(* ---------------------- Debug-Message ----------------------------*)
(*IF  _debug_enable THEN
	IF state <> state_last THEN
		LOG_CL.NEW_MSG := 'IP_STEP ~1 -IP_ID ~6';
		LOG_CL.PRINTF[1] := BYTE_TO_STRING(state);
		LOG_CL.PRINTF[6] := INT_TO_STRING(debug_ID);
		LOG_MSG();
		state_last := state;
	END_IF;
END_IF;*)
(* -----------------------------------------------------------------------------*)

IF IP_C.TIME_RESET THEN (* Alle Timer ruecksetzen *)
	IP_C.TIME_RESET := FALSE; (* Reset rücksetzen *)
	c_time := tx; (* Connect Timer ruecksetzen *)
	s_time := tx; (* Send Timer ruecksetzen *)
	r_time := tx; (* Receive Timer ruecksetzen *)

	c_status := BYTE#0; (* letzten Connect Fehler rücksetzen *)
	s_status := BYTE#0; (* letzten Send Fehler rücksetzen *)
	r_status := BYTE#0; (* letzten Receive Fehler rücksetzen *)
END_IF;

(* ---------------------------------------------- *)

CASE state OF

UDP_INIT: (* UDP_CLIENT + SERVER *)
	socket := SysSockCreate(SOCKET_AF_INET, SOCKET_DGRAM, SOCKET_IPPROTO_IP, ADR(pResult));
	IF socket < 0 THEN
		c_status := 1; (* SysSockCreate failed *)
		state := C_CLOSE;
	ELSE
		FunctionResult :=SysSockSetOption(socket, SOCKET_SOL, SOCKET_SO_BROADCAST, ADR(dint_true), SIZEOF(dint_true)); (* allow broadcast *)
		FunctionResult :=SysSockIoctl(socket, SOCKET_FIONBIO, ADR(dint_true)); (* put socket in non-blocking mode *)
		sockaddr.sin_family := SOCKET_AF_INET;
		sockaddr.sin_port := SysSockHtons(c_port);
		sockaddr.sin_addr.ulAddr := SEL(c_mode = 1, SOCKET_INADDR_ANY, SysSockNtohl(c_ip));

		IF c_mode >= 2 THEN (* SERVER Mode *)
			FunctionResult := SysSockBind(socket, ADR(sockaddr), SIZEOF(sockaddr));
			IF FunctionResult=0 THEN
				c_ready := TRUE; (* Connected *)
				state:= C_WAIT;
			ELSE
				c_status := 2; (* SysSockBind failed *)
				state := C_CLOSE;
			END_IF;
		ELSE
			c_ready := TRUE; (* Connected *)
			state:= C_WAIT;
		END_IF;
	END_IF;

(* ---------------------------------------------- *)

TC_INIT: (* TCP-CLIENT (AKTIV) *)
	// Create handle to ethernet socket to send messages
	socket        := SysSockCreate(SOCKET_AF_INET, SOCKET_STREAM, SOCKET_IPPROTO_TCP, ADR(pResult)); 	
	IF socket < 0 THEN
		c_status := 1;  (* SysSockCreate failed *)
		state := C_CLOSE;
	ELSE
		IF plc_841 OR plc_881 THEN
			FunctionResult :=SysSockSetOption(socket,6,SOCKET_TCP_NODELAY, ADR(dint_true), SIZEOF(dint_true)); (* Set Push-Bit *)
		END_IF;
		// Set option for local address reuse
		FunctionResult :=SysSockSetOption(socket, SOCKET_SOL, SOCKET_SO_REUSEADDR, ADR(dint_true), SIZEOF(dint_true));
		// Set option for keepalive
		//FunctionResult := SysSockSetOption(socket, SOCKET_SOL, SOCKET_SO_KEEPALIVE, ADR(dint_true), SIZEOF(dint_true));
		
        FunctionResult :=SysSockIoctl(socket, SOCKET_FIONBIO, ADR(dint_true)); (* NonBlocking mode *)
		
		sockaddr.sin_family := SOCKET_AF_INET;
		sockaddr.sin_port := SysSockNtohs(c_port);
		sockaddr.sin_addr.ulAddr  := SysSockNtohl(c_ip);
		c_select := FALSE;
		state := TC_CONNECT;
	END_IF;

(* ---------------------------------------------- *)

TC_CONNECT:
	IF NOT c_enable OR c_status = 255 THEN (* keine freigabe oder connect timeout *)
			state:= C_CLOSE;
	ELSE
		IF c_select = FALSE THEN
			FunctionResult:=SysSockConnect(socket,ADR(sockaddr),SIZEOF(sockaddr));
			IF FunctionResult=0 THEN
				c_ready := TRUE; (* Connected *)
				state:= C_WAIT;
			ELSE
				(* Connect durchgeführt, aber noch nicht verbunden, dann optional mit select-abfrage weitermachen *)
				c_select := SYSLIBSOCKETS_OPTION.0; (* Bit 0 = TCP-Client - use SysSockselect *)
			END_IF;
		ELSE
			c_Timeout.tv_sec := 0;
			c_Timeout.tv_usec := 0;
			c_fdWrite.fd_count := 1;
			c_fdWrite.fd_array[0] := socket;
			IF SysSockSelect(SOCKET_FD_SETSIZE,0,ADR(c_fdWrite),0, ADR(c_Timeout), ADR(pResult)) > 0 THEN
				c_ready := TRUE; (* Connected *)
				state:= C_WAIT;
			END_IF;
		END_IF;
	END_IF;

(* ---------------------------------------------- *)

TS_INIT: (* TCP-SERVER (PASSIV) *)
	server_socket := SysSockCreate(SOCKET_AF_INET, SOCKET_STREAM, SOCKET_IPPROTO_IP, ADR(pResult)); (* Create Socket *)
	IF server_socket = RTS_INVALID_HANDLE THEN
		c_status := 1; (* SysSockCreate failed *)
		state:= C_CLOSE;
	ELSE (* Address bindings *)
		SysSockSetOption( server_socket, SOCKET_SOL, SOCKET_SO_REUSEADDR, ADR(dint_true), SIZEOF(dint_true) );
		sockaddr.sin_family:= SOCKET_AF_INET;
		sockaddr.sin_port := SysSockHtons(c_port);
		sockaddr.sin_addr.ulAddr  := SOCKET_INADDR_ANY;
		IF NOT SysSockBind(server_socket, ADR(sockaddr), SIZEOF(sockaddr)) = 0 THEN
			c_status := 2; (* SysSockBind failed *)
			state := C_CLOSE;
		ELSIF NOT SysSockListen(server_socket, 1) = 0 THEN (* erzeugt Warteschlange für eine Verbindung *)
			c_status := 3; (* SysSockListen failed *)
			state:= C_CLOSE;
		ELSE
			SysSockIoctl(server_socket, SOCKET_FIONBIO, ADR(dint_true)); (* NonBlocking mode *)
			state:= TS_OPEN;
		END_IF;
	END_IF;

(* ---------------------------------------------- *)

TS_OPEN: (* Waiting for incomming connection *)
	sockaddr_size := SIZEOF(sockaddr);
	socket := SysSockAccept(server_socket, ADR(sockaddr), ADR(sockaddr_size), ADR(pResult));

	IF socket <> RTS_INVALID_HANDLE THEN (* neuer Verbindungswunsch vorhanden *)
		IF c_mode = BYTE#2 AND sockaddr.sin_addr.ulAddr <> SysSockNtohl(c_ip) THEN (* Mode 2 = TCP + PASSIVE + PORT + IP  auf richtige Partner-IP prüfen *)
			state:= C_CLOSE;
		ELSE
			IF plc_841 OR plc_881 THEN
				SysSockSetOption(socket, 6, SOCKET_TCP_NODELAY, ADR(dint_true), SIZEOF(dint_true)); (* Set Push-Bit *)
			END_IF;
			SysSockIoctl(socket, SOCKET_FIONBIO, ADR(dint_true)); (* NonBlocking mode *)
			c_ready := TRUE; (* Connected *)
			state := C_WAIT;
		END_IF;
	ELSIF NOT c_enable THEN (* keine freigabe mehr ? *)
			state:= C_CLOSE;
	END_IF;

(* ---------------------------------------------- *)

C_WAIT: (* Warten auf Anforderung für Beenden *)
	IF NOT c_enable OR NOT c_ready THEN
		state:= C_CLOSE;
	END_IF

(* ---------------------------------------------- *)

C_CLOSE: (* Close the Sockets *)
	c_ready := FALSE;
	IF socket >= 0 THEN
		IF (NOT plc_841) AND (NOT plc_881) THEN
			SysSockShutdown(socket, 0); (* 870 *)
		END_IF;
		SysSockClose(socket);
		socket := RTS_INVALID_HANDLE;
	END_IF
	IF server_socket >= 0 THEN
		IF (NOT plc_841) AND (NOT plc_881) THEN
			SysSockShutdown(server_socket, 0); (* 870 *)
		END_IF;
		SysSockClose(server_socket);
		server_socket := RTS_INVALID_HANDLE;
	END_IF
	state:= STOP;
END_CASE;

(* ---------------------------------------------- *)

IF c_ready THEN
	IF NOT c_ready_old THEN (* Verbindung aufgebaut - positive Flanke erkannt *)
		IP_C.C_STATE := 254;
		IP_C.TIME_RESET := TRUE; (* Alle Timer ruecksetzen *)
		(* ---------------------- Debug-Message ----------------------------*)
		(*IF _debug_enable THEN
			LOG_CL.NEW_MSG := 'IP_CON: CONNECTED -IP_ID ~6';
			LOG_CL.PRINTF[6] := INT_TO_STRING(debug_ID);
			LOG_MSG();
		END_IF;*)
		(* -----------------------------------------------------------------------------*)
	ELSE
		IP_C.C_STATE := 255; (* Verbindung ist aufgebaut *)
	END_IF;
ELSE
	IF c_ready_old THEN (* Verbindung abgebaut - negative Flanke erkannt *)
		IP_C.C_STATE := 1;
		IP_C.MAILBOX[1] := 0; (* Receive Info rücksetzen *)
		IP_C.MAILBOX[2] := 0; (* Send-Pause rücksetzen *)
		IP_C.MAILBOX[3] := 0; (* Receive-Pause rücksetzen *)
		IF NOT new_connection THEN
			s_active := FALSE; (* Sendeaktivitäten stoppen *)
			s_req := FALSE; (* Sendefreigabe rücksetzen *)
			S_BUF.SIZE := 0; (* Sendelänge löschen *)
			(*IP_C.TIME_RESET := TRUE;*) (* Alle Timer ruecksetzen *)
		END_IF;
		(* ---------------------- Debug-Message ----------------------------*)
		(*IF _debug_enable THEN
			LOG_CL.NEW_MSG := 'IP_CON: DISCONNECTED';
			LOG_MSG();
		END_IF;*)
		(* -----------------------------------------------------------------------------*)
	ELSE
		IP_C.C_STATE := 0; (* Verbindung ist abgebaut *)
	END_IF;
END_IF;

c_ready_old := c_ready;

(* Der Datenempfang wird angehalten solange ein Sendevorgang läuft *)
(* sonst kann es vorkommen das die Antwort-daten schon empfangen werden, *)
(* bevor der Sendevorgang vom programm abgeschlossen wurde *)

IF c_ready AND NOT s_active AND IP_C.MAILBOX[3] = 0 THEN
	IF R_BUF.SIZE >= INT_TO_UINT(r_max_size) THEN
		R_BUF.SIZE := UINT#0;
		r_status := 254; (* Empfangsbuffer wegen Überlauf rückgesetzt *)
	END_IF;

	r_offset := SEL(udp_mode,UINT_TO_INT(R_BUF.SIZE),0);
	r_count := r_max_size - r_offset;

	IF udp_mode THEN
		bytes_received := SysSockRecvFrom(socket, ADR(R_BUF.BUFFER), r_count, 0, ADR(sockaddr), SIZEOF(sockaddr), ADR(pResult));

		IF c_mode = BYTE#3 AND sockaddr.sin_addr.ulAddr <> SysSockNtohl(c_ip) THEN (* Mode 3 = UDP + PASSIVE + PORT + IP  auf richtige Partner-IP prüfen *)
			bytes_received := 0;
			R_BUF.SIZE := UINT#0;
			sockaddr.sin_port := SysSockNtohs(c_port);
			sockaddr.sin_addr.ulAddr  := SysSockNtohl(c_ip);
		END_IF;

	ELSE
		bytes_received := SysSockRecv(socket, ADR(R_BUF.BUFFER[r_offset]), r_count, 0, ADR(pResult));
	END_IF;

	CASE pResult OF
		518:  bytes_received:=-1; //Connection OKAY just no data and do not want to BIND
		521:  bytes_received:=0; //Connection has been refused by the remote host 
		523:  bytes_received:=0; //The host has not been found  
		524:  bytes_received:=0; //Host is unreachable  
		526:  bytes_received:=0; //The socket is not connected  
		527:  bytes_received:=0; //Shutdown has been called on the socket  
		529:  bytes_received:=0; //Socket has been gracefully closed. No more send/receives allowed	 
	END_CASE

	
	(*UDP: IPC returns -1 if no data available or error occured,841 returns -1 if error occured and 0 if no data available*)
	CASE bytes_received OF
	-2147483648..-1: ; (* No data available or error occured *)
	 0: IF NOT udp_mode OR pResult<>518 THEN (* TCP-Mode: socket wurde von remote geschlossen *)
			c_status := 253;
			c_ready := FALSE;
		END_IF;
	ELSE (* daten wurden empfangen *)
  		r_time := tx; (* Receive Timer ruecksetzen *)
		R_BUF.SIZE := INT_TO_UINT(r_offset) + DINT_TO_UINT(bytes_received); (* aktuelle buffersize eintragen *)
		IP_C.MAILBOX[1] := IP_C.MAILBOX[1] + 1; (* Receive Info *)
		IF IP_C.MAILBOX[1] = 0 THEN IP_C.MAILBOX[1] := 1; END_IF;

		(* ---------------------- Debug-Message ----------------------------*)
		(*IF _debug_enable THEN
			LOG_CL.NEW_MSG := 'IP_REC DATA: POS: ~1 : SIZE: ~2 TOTAL ~3 -IP_ID ~6';
			LOG_CL.PRINTF[1] := INT_TO_STRING(r_offset);
			LOG_CL.PRINTF[2] := INT_TO_STRING(r_count);
			LOG_CL.PRINTF[3] := UINT_TO_STRING(R_BUF.SIZE);
			LOG_CL.PRINTF[6] := INT_TO_STRING(debug_ID);
			LOG_MSG();
		END_IF;*)
		(* -----------------------------------------------------------------------------*)

	END_CASE
END_IF;

(* ---------------------------------------------- *)

IF S_BUF.SIZE > 0 THEN
	IF c_ready AND c_enable THEN
		IF NOT s_active AND IP_C.MAILBOX[2] = 0 THEN
			(* Gesamtanzahl an Bytes limitieren und uebergeben *)
			s_total := LIMIT(0,UINT_TO_INT(S_BUF.SIZE),r_max_size);
			s_cur_pos  := 0;
			s_cur_size := 0;
			s_start := TRUE; (* Daten kopieren und senden anstossen *)
			s_active := TRUE; (* Sende-Betrieb aktivieren *)
			(* ---------------------- Debug-Message ----------------------------*)
			(*IF _debug_enable THEN
				LOG_CL.NEW_MSG := 'IP_SEN INIT: TOTAL: ~1 -IP_ID ~6';
				LOG_CL.PRINTF[1] := INT_TO_STRING(S_TOTAL);
				LOG_CL.PRINTF[6] := INT_TO_STRING(debug_ID);
				LOG_MSG();
			END_IF;*)
			(* -----------------------------------------------------------------------------*)
		END_IF;

		IF s_done OR s_start THEN (* Daten senden aktiv *)

			s_start := FALSE;
			s_cur_pos := s_cur_pos + s_cur_size; (* neue Sende-Datenposition bestimmen *)
			IF s_total > s_cur_pos THEN (* weitere Daten zum senden vorhanden ? *)
				s_cur_size := s_total - s_cur_pos;
				s_cur_size := LIMIT(0, s_cur_size, s_max_size); (* Telegrammlänge begrenzen *)
				(* ---------------------- Debug-Message ----------------------------*)
				(*IF _debug_enable THEN
					LOG_CL.NEW_MSG := 'IP_SEN DATA: POS: ~1 : SIZE: ~2 TOTAL ~3 -IP_ID ~6';
					LOG_CL.PRINTF[1] := INT_TO_STRING(S_CUR_POS);
					LOG_CL.PRINTF[2] := INT_TO_STRING(S_CUR_SIZE);
					LOG_CL.PRINTF[3] := INT_TO_STRING(S_TOTAL);
					LOG_CL.PRINTF[6] := INT_TO_STRING(debug_ID);
					LOG_MSG();
				END_IF;*)
				(* -----------------------------------------------------------------------------*)
				s_time := tx; (* Send Timer ruecksetzen *)
				r_time := tx; (* Receive Timer ruecksetzen *)
				s_req := TRUE;

			ELSE
				(* keine weitere Sendedaten vorhanden -> Senden beenden *)
				s_req := FALSE;
				s_active := FALSE;
				S_BUF.SIZE := 0;
				(* ---------------------- Debug-Message ----------------------------*)
				(*IF _debug_enable THEN
					LOG_CL.NEW_MSG := 'IP_SEN FINISH -IP_ID ~6';
					LOG_CL.PRINTF[6] := INT_TO_STRING(debug_ID);
					LOG_MSG();
				END_IF;*)
				(* -----------------------------------------------------------------------------*)
			END_IF;
		END_IF;
	END_IF;
END_IF;

IF s_req THEN
	s_done := FALSE;
	IF udp_mode THEN
		bytes_sent := SysSockSendTo(socket, ADR(S_BUF.BUFFER[s_cur_pos]), s_cur_size, 0, ADR(sockaddr), SIZEOF(sockaddr), ADR(pResult));
	ELSE
		bytes_sent := SysSockSend(socket, ADR(S_BUF.BUFFER[s_cur_pos]), s_cur_size, 0, ADR(pResult));
	END_IF;

	CASE bytes_sent OF
	-2147483648..-1:	; (* ERROR: Noch nicht bereit um Daten aufzunehmen -> nächsten Zyklus wieder probieren *)
	 0: IF NOT udp_mode THEN (* TCP-Mode: socket wurde von remote geschlossen *)
			c_status := 253;
			c_ready := FALSE;
		END_IF;
	ELSE
		s_done := TRUE;
		s_cur_size := DINT_TO_INT(bytes_sent); (* Anzahl der wirklich versendeten Bytes übernehmen *)
		(* ---------------------- Debug-Message ----------------------------*)
		(*IF _debug_enable THEN
			LOG_CL.NEW_MSG := 'IP_SEN SEND_COUNT ~1 -IP_ID ~6';
			LOG_CL.PRINTF[1] := DINT_TO_STRING(s_cur_size);
			LOG_CL.PRINTF[6] := INT_TO_STRING(debug_ID);
			LOG_MSG();
		END_IF;*)
		(* -----------------------------------------------------------------------------*)
	END_CASE
END_IF;

(* ---------------------------------------------- *)

IF IP_C.R_OBSERVE = FALSE OR s_active THEN
    r_time := tx;
END_IF;

IF c_status = 0 AND tx - c_time > error_time AND c_enable AND NOT c_ready AND c_mode < 2 THEN (* Connect Timeout *)
	c_status := 255; (* Timeout-Fehler ausgeben *)
END_IF;
IF s_status = 0 AND tx - s_time > error_time AND s_active THEN (* Send Timeout *)
	s_status := 255; (* Timeout-Fehler ausgeben *)
END_IF;
IF r_status = 0 AND tx - r_time > error_time AND c_ready AND IP_C.R_OBSERVE THEN (* Receive Timeout *)
	r_status := 255; (* Timeout-Fehler ausgeben *)
END_IF;

IP_C.ERROR := OSCAT_BASIC.DWORD_OF_BYTE(c_status,s_status,r_status,0);

(* ---------------------- Debug-Message ----------------------------*)
(*IF  _debug_enable THEN
	IF (IP_C.ERROR <> debug_lasterror) THEN
		LOG_CL.NEW_MSG := 'IP_ERROR ~1 -IP_ID ~6';
		LOG_CL.PRINTF[1] := DWORD_TO_STRING(IP_C.ERROR);
		LOG_CL.PRINTF[6] := INT_TO_STRING(debug_ID);
		LOG_MSG();

		debug_lasterror := IP_C.ERROR;
		debug_last_id := debug_ID;
	END_IF;
END_IF;*)
(* -----------------------------------------------------------------------------*)

(* revision history
ks	18. oct. 2008	rev 1.0
	original version
ks	05. jan. 2009	rev 1.1
	zusätzlichen Parameter "Port" hinzugefügt, und Code bei Verbindungsaufbau angepasst
ks	28. feb. 2009	rev 1.2
	connect code angepasst und verkürzung der zyklen bei Send
ks	20. oct. 2009	rev 1.3
	network_buffer basis 0
ks	06. dec. 2009	rev 1.4
	receive_count MAILBOX[1]
ks	10. nov. 2010	rev 1.5
	send_pause MAILBOX[2] and receive_pause MAILBOX[3] 
ks	07. feb. 2011	rev 1.6
	Fehlercode 253 bei Remote-Verbindungsabbruch
ks	30. may. 2011	rev 1.7
	Fehler bei Empfangsüberwachung
ks	26. july. 2011	rev 1.8
	Error-Reset, diverse optimierungen 
ks	26. feb. 2012	rev 1.9
	Code-Optimierung für höhere kompatibilität

*)

END_FUNCTION_BLOCK

// Common/Function Blocks/TIME_DATE_IMPULS
FUNCTION_BLOCK TIME_DATE_IMPULS
VAR_IN_OUT
	TDI_Data:TIME_DATE_IMPULS_DATA;
END_VAR
VAR_INPUT
END_VAR

VAR
	RT_SYS:RTCLK.GetDateAndTime;
	RT:OSCAT_BASIC.RTC_2;
	DT_OLD:DT;
	GET_TIME: BOOL := TRUE;
	TIME_READED: BOOL;
	TIMEZONE:RTCLK.PERIODE;
	ReReadTime: BOOL;
	ReReadErrorTime:TON;
	ReReadTimeCycle:TON;
	DayChangeEdge:R_TRIG;
END_VAR

RT_SYS(xExecute := GET_TIME);
IF RT_SYS.xDone THEN
	GET_TIME := FALSE;
	IF	RT_SYS.dtDateAndTime < DT#1980-01-01-00:00:00 THEN
		//Keine Valide Uhr auf Raspi!
		ReReadTime := TRUE;
		TDI_Data.TIME_IO := FALSE;
	ELSE
		TIME_READED := TRUE;
		TIMEZONE := RT_SYS.eTimezone;
		ReReadTime := FALSE;
		TDI_Data.TIME_IO := TRUE;
	END_IF
END_IF
//Zykliches neulsesen der Uhrzeit
ReReadTimeCycle(in := (TDI_Data.TIME_IO AND NOT GET_TIME), PT:= T#30M);
IF ReReadTimeCycle.Q THEN
	GET_TIME := TRUE;//try again to read Time	
END_IF


//Neulesezeit nach Error bearbeiten:
ReReadErrorTime(in:=ReReadTime, pt:=T#1S);
IF ReReadErrorTime.Q THEN
	ReReadTime := FALSE;
	GET_TIME := TRUE;//try again to read Time
END_IF
//Realtime Clock bearbeiten // Setzten
RT(set := TIME_READED, SDT := RT_SYS.dtDateAndTime, OFS := 60, DEN:=TRUE,);
TIME_READED := FALSE;
//Date and time from oscat fb
TDI_Data.SYSTEM_TIME:=RT._LDT;
//check for second impuls
IF DT_OLD <> TDI_Data.SYSTEM_TIME THEN
	DT_OLD := TDI_Data.SYSTEM_TIME;
	TDI_Data.imp := TRUE;
ELSE
	TDI_Data.imp := FALSE;
END_IF
//make Time for OSCAT functions
TDI_Data.TD_TIME := OSCAT_BASIC.DT_TO_SDT(DTI:= TDI_Data.SYSTEM_TIME);
TDI_Data.UDT := RT.UDT;

DayChangeEdge(CLK:=TO_TOD(TDI_DATA.SYSTEM_TIME)= TOD#00:00:00);
TDI_DATA.DAY_CHANGE := DayChangeEdge.Q;

END_FUNCTION_BLOCK

// Common/Functions/GET_DNS_IP
FUNCTION GET_DNS_IP : STRING(16)
VAR_INPUT
END_VAR
VAR
	Result:RTS_IEC_RESULT;
	DNS_STRING:STRING(1000);
	findRet:DINT;
	i:INT;
	j:INT;
	k:INT;
	start:INT;
	stop:INT;
	//id of operating system
	OsId:UDINT;
END_VAR
VAR CONSTANT
	GET_DNS_COMMAND_LINUX:STRING:='cat /etc/resolv.conf ';//|grep -i nameserver|head -n1|cut -d $' $' -f2';
	GET_DNS_COMMAND_WINDOWS:STRING:='powershell Get-DnsClientServerAddress';//|grep -i nameserver|head -n1|cut -d $' $' -f2';
	NAMESERVER_LINUX:STRING:='nameserver';
	
END_VAR

(*
for linux

change 
sudo nano /etc/CODESYSControl.cfg
or from runtime version 4.5.11.20
sudo nano /etc/CODESYSControl_User.cfg 
[SysProcess]
Command.0=shutdown

to 

[SysProcess]
Command.0=shutdown
Command.1=cat

for windows, needs powershell

"C:\ProgramData\CODESYS\CODESYSControlWinV3\???\CODESYSControl.cfg"
[SysProcess]
BasePriority=Realtime
Command=AllowAll

*)

//cat /etc/resolv.conf |grep -i nameserver|head -n1|cut -d ' ' -f2
//get content

SysTargetGetOperatingSystemId(pudiOperatingSystemId:= ADR(OsId));


GET_DNS_IP := 'ERROR';

IF OsId = OperatingSystemID.SYSTARGET_OS_LINUX THEN

	SysProcess.SysProcessExecuteCommand2(pszCommand:=GET_DNS_COMMAND_LINUX,pszStdOut:= DNS_STRING,udiStdOutLen:=SIZEOF(DNS_STRING),pResult:=ADR(Result));
	IF Result = CmpErrors.Errors.ERR_NO_ACCESS_RIGHTS THEN
		GET_DNS_IP := 'NOACCESSRIGHTS';
		RETURN;
	END_IF
	//TODO check if command is enabled 
	i:= Standard.FIND(STR1:=DNS_STRING, STR2:=NAMESERVER_LINUX);
	IF i < 0 THEN RETURN; END_IF
	j := OSCAT_BASIC.FIND_CTRL(str:= DNS_STRING, pos:= i);
	IF j <= 0 THEN RETURN; END_IF
	
	GET_DNS_IP := Standard.MID(STR:= DNS_STRING, LEN:= j - i - Standard.LEN(STR:=NAMESERVER_LINUX) - 1, POS:= i + Standard.LEN(NAMESERVER_LINUX) + 1);
	
END_IF

IF OsId = OperatingSystemID.SYSTARGET_OS_WINDOWS THEN
{info 'TODO: hind that this is blocking!'}
SysProcess.SysProcessExecuteCommand2(pszCommand:=GET_DNS_COMMAND_WINDOWS,pszStdOut:= DNS_STRING,udiStdOutLen:=SIZEOF(DNS_STRING),pResult:=ADR(Result));
	IF Result = CmpErrors.Errors.ERR_NO_ACCESS_RIGHTS THEN
		GET_DNS_IP := 'NOACCESSRIGHTS';
		RETURN;
	END_IF
	//TODO check if command is enabled 
	findRet:= find(STR1:=ADR(DNS_STRING), STR2:=ADR('IPv4'));
	IF findRet < 0 THEN RETURN; END_IF
	i := DINT_TO_INT(findRet);
	//now search '{'
	FOR j := 0 TO 40 DO//max 40 chars space
		IF DNS_STRING[i + j] = GetChar('{') THEN
			start := i + j + 1;
		END_IF
 		IF DNS_STRING[i + j] = GetChar('}') THEN
			stop := i + j - 1;
			EXIT;
		END_IF
	END_FOR
	//now copy data, string functions usless --> more than 255 chars...
	
	j := 0;
	FOR i := start TO stop DO
		GET_DNS_IP[j] := DNS_STRING[i];
		j := j + 1;
	END_FOR
	GET_DNS_IP[j] := 0;//termination
	
	//j := OSCAT_BASIC.FIND_CTRL(str:= DNS_STRING, pos:= i);
//	IF j <= 0 THEN RETURN; END_IF
	
	//GET_DNS_IP := Standard.MID(STR:= DNS_STRING, LEN:= j - i - Standard.LEN(STR:=NAMESERVER_LINUX) - 1, POS:= i + Standard.LEN(NAMESERVER_LINUX) + 1);
	

END_IF

END_FUNCTION

// Common/Functions/find
//searchs str2 in str1
FUNCTION find : DINT
VAR_INPUT
	str1:POINTER TO STRING;
	str2:POINTER TO STRING;
END_VAR
VAR
	
	n:UINT;	
	pt:POINTER TO BYTE;
	
	j: UINT;
END_VAR

find := -1;//first we din't find anything....
n := len(str := str2);


pt := str1;

WHILE pt^ <> 0 DO
	IF SysMemCmp(pBuffer1:= pt, pBuffer2:= str2, udiCount:= n) = 0 THEN
		
		find := j;
		RETURN;
	
	END_IF
	j := j + 1;
	pt := pt + SIZEOF(BYTE);
	
END_WHILE

END_FUNCTION

// Common/Functions/len
FUNCTION len : UINT
VAR_INPUT
	str:POINTER TO STRING;
END_VAR
VAR
	k:uINT;
	pt:POINTER TO BYTE;
END_VAR

pt := str;
WHILE pt[k] <>  0 DO
	k := k + 1;
END_WHILE
len := k;

END_FUNCTION

// Common/Functions/GetChar
FUNCTION GetChar : byte
VAR_INPUT
	in:STRING(1);
END_VAR

GetChar := in[0];

END_FUNCTION

// Common/Functions/concat
FUNCTION concat : pointer to string
VAR_INPUT
	s1:POINTER TO STRING;
	s2:POINTER TO STRING;
END_VAR
VAR
	p1:POINTER TO BYTE;
	len1:UINT;
	
	ui:UINT;
END_VAR

p1 := ADR(s1^[len(s1)]);
len1 := len(s2);
SysMemMove(pDest:= p1, pSrc:= s2, udiCount:= len1 + 1);//+ 1 for add 0 to string end

concat := s1;

END_FUNCTION

// Common/Function Blocks/TestString
FUNCTION_BLOCK TestString 
VAR_INPUT
END_VAR
VAR
	s10:STRING:='1111111111';
	s102:STRING:='2222222222';
	sp:STRING(64000);
	ps1:POINTER TO STRING;
	lens:UINT;
END_VAR

lens := len(ADR(s10)); //needs to be 10!
sp:='';
concat(s1:= ADR(sp), s2:= ADR(s10));
ps1 := ADR(sp);
lens := len(ADR(sp)); //needs to be 10!

concat(s1:= ADR(sp), s2:= ADR(s102));

lens := len(ADR(sp)); //needs to be 20!

concat(s1:= ADR(sp), s2:= ADR(s10));

lens := len(ADR(sp)); //needs to be 30!

concat(s1:= ADR(sp), s2:= ADR(s102));

lens := len(ADR(sp)); //needs to be 40!

concat(s1:= ADR(sp), s2:= ADR(s10));

lens := len(ADR(sp)); //needs to be 50!

concat(s1:= ADR(sp), s2:= ADR(sp));

lens := len(ADR(sp)); //needs to be 100!

concat(s1:= ADR(sp), s2:= ADR(sp));

lens := len(ADR(sp)); //needs to be 200!

concat(s1:= ADR(sp), s2:= ADR(sp));

lens := len(ADR(sp)); //needs to be 400!

concat(s1:= ADR(sp), s2:= ADR(sp));

lens := len(ADR(sp)); //needs to be 800!

concat(s1:= ADR(sp), s2:= ADR(sp));

lens := len(ADR(sp)); //needs to be 1600!

concat(s1:= ADR(sp), s2:= ADR(sp));

lens := len(ADR(sp)); //needs to be 3200!

concat(s1:= ADR(sp), s2:= ADR(sp));

lens := len(ADR(sp)); //needs to be 6400!

END_FUNCTION_BLOCK

// Common/Function Blocks/IP_CONTROL_TLS
FUNCTION_BLOCK IP_CONTROL_TLS EXTENDS IP_CONTROL
VAR_INPUT
	TLS_CONFIG_IN:POINTER TO TLS_CONFIG := 0;(*info about tls stuff*)
	useTls: BOOL;

END_VAR
VAR_OUTPUT
END_VAR
VAR
	
END_VAR


TLS:= useTls;
IF TLS THEN
	TLS_CONFIG := TLS_CONFIG_IN;
END_IF
SUPER^(IP_C := IP_C, R_BUF:= R_BUF, S_BUF:= S_BUF);

END_FUNCTION_BLOCK

// Common/Functions/ResolveIPAddr
/// This function resolves the IP of the domain name. 
FUNCTION ResolveIPAddr : RTS_IEC_RESULT
VAR_INPUT
	sHost : STRING;
	sIPResult : POINTER TO STRING; 
END_VAR
VAR
	refsHost : REFERENCE TO STRING := sHost;
	stSockHost : SOCK_HOSTENT;
	rtsResultSock : RTS_IEC_RESULT;
	rtsResultInAddr : RTS_IEC_RESULT;
	stinAddr : INADDR;
	ptdwHostAddr : POINTER TO __XWORD;
	dwHostAddr : __XWORD;
	sServerIP : STRING;
END_VAR

rtsResultSock := SysSockGetHostByName(refsHost,ADR(stSockHost));
IF rtsResultSock = CmpErrors.Errors.ERR_OK THEN
	ptdwHostAddr := stSockHost.pAddrList[0]; // Eth Adapter
	dwHostAddr := ptdwHostAddr^;
	IF dwHostAddr <> SOCKET_INADDR_NONE THEN
		stinAddr.ulAddr := __XWORD_TO_UDINT(dwHostAddr);
		rtsResultInAddr := SysSockInetNtoa(pInAddr:=ADR(stinAddr),szIPADDR:=sServerIP ,diIPAddrSize:=SIZEOF(sServerIP));
		IF rtsResultInAddr = CmpErrors.Errors.ERR_OK THEN
			sIPResult^ := sServerIP;
		ELSE
			ResolveIPAddr := CmpErrors.Errors.ERR_FAILED;
		END_IF
	END_IF
ELSE
	ResolveIPAddr := CmpErrors.Errors.ERR_FAILED;
END_IF

END_FUNCTION

// Common/Functions/CheckDeltaValue
FUNCTION CheckDeltaValue : bool
VAR_INPUT
	Value:ALL_TYPES_UNION;
	TypeOfValue:VAR_TYPES;
	DeltaVar:UINT;
	Faktor:UINT;
END_VAR
VAR_IN_OUT
	LastValue:ALL_TYPES_UNION;
END_VAR
VAR
END_VAR

(*	SINT_T, USINT_T, INT_T, UINT_T, DINT_T, UDINT_T, 
				LINT_T, ULINT_T, REALT_T, LREAL_T*)
CASE TypeOfValue OF
	VAR_TYPES.SINT_T:
		//CheckDeltaValue := (ABS(LAST_VALUE.SINT_T) + UINT_TO_SINT(DELTA_VAR)) > ABS(Value.SINT_T);
		CheckDeltaValue := ABS(LastValue.SINT_T - Value.SINT_T) >= UINT_TO_SINT(DeltaVar);
		
		IF CheckDeltaValue THEN LastValue.SINT_T := Value.SINT_T; END_IF
	VAR_TYPES.USINT_T:

		CheckDeltaValue := ABS(USINT_TO_INT(LastValue.USINT_T) - USINT_TO_INT(Value.USINT_T)) >= UINT_TO_USINT(DeltaVar);
		IF CheckDeltaValue THEN LastValue.USINT_T := Value.USINT_T; END_IF
	VAR_TYPES.INT_T:
		CheckDeltaValue := ABS(LastValue.INT_T - Value.INT_T) >= + UINT_TO_INT(DeltaVar);
		IF CheckDeltaValue THEN LastValue.INT_T := Value.INT_T; END_IF
	VAR_TYPES.UINT_T:
		CheckDeltaValue := ABS(UINT_TO_DINT(LastValue.UINT_T) - UINT_TO_DINT(Value.UINT_T)) >= DeltaVar;
		IF CheckDeltaValue THEN LastValue.UINT_T := Value.UINT_T; END_IF
	VAR_TYPES.DINT_T:
		CheckDeltaValue := ABS(LastValue.DINT_T - Value.DINT_T) >= + UINT_TO_DINT(DeltaVar);
		IF CheckDeltaValue THEN LastValue.DINT_T := Value.DINT_T; END_IF
	VAR_TYPES.UDINT_T:
		CheckDeltaValue := ABS(UDINT_TO_LINT(LastValue.UDINT_T) - UDINT_TO_LINT(Value.UDINT_T)) >= DeltaVar;
		IF CheckDeltaValue THEN LastValue.UDINT_T := Value.UDINT_T; END_IF
	VAR_TYPES.LINT_T:
		CheckDeltaValue := ABS(LastValue.LINT_T - Value.LINT_T) >= + UINT_TO_LINT(DeltaVar);
		IF CheckDeltaValue THEN LastValue.LINT_T := Value.LINT_T; END_IF
	VAR_TYPES.ULINT_T:
	//here we use no expand but check min max because no bigger data type...
		IF LastValue.ULINT_T <= Value.ULINT_T THEN
			CheckDeltaValue := Value.ULINT_T - LastValue.ULINT_T >= UINT_TO_ULINT(DeltaVar);	
		ELSE
			CheckDeltaValue := LastValue.ULINT_T - Value.ULINT_T >= UINT_TO_ULINT(DeltaVar);
		END_IF
		IF CheckDeltaValue THEN LastValue.ULINT_T := Value.ULINT_T; END_IF
	VAR_TYPES.REAL_T:
		CheckDeltaValue := ABS(LastValue.REAL_T * Faktor - Value.REAL_T * Faktor) >= UINT_TO_REAL(DeltaVar)  ;
		IF CheckDeltaValue THEN LastValue.REAL_T := Value.REAL_T; END_IF
	VAR_TYPES.LREAL_T:
		//CheckDeltaValue := (ABS(LAST_VALUE.LREAL_T * RealFaktor) + UINT_TO_LREAL(DeltaVar)) <= ABS(Value.LREAL_T * RealFaktor);
		CheckDeltaValue := ABS(LastValue.LREAL_T * Faktor - Value.LREAL_T * Faktor) >= UINT_TO_LREAL(DeltaVar)  ;
		IF CheckDeltaValue THEN LastValue.LREAL_T := Value.LREAL_T; END_IF
	VAR_TYPES.BYTE_T:
		CheckDeltaValue := ABS(BYTE_TO_INT(LastValue.BYTE_T) - BYTE_TO_INT(Value.BYTE_T)) >= UINT_TO_INT(DeltaVar);
		IF CheckDeltaValue THEN LastValue.BYTE_T := Value.BYTE_T; END_IF
	VAR_TYPES.WORD_T:
		CheckDeltaValue := ABS(WORD_TO_DINT(LastValue.WORD_T) - WORD_TO_DINT(Value.WORD_T)) >= DeltaVar;
		IF CheckDeltaValue THEN LastValue.WORD_T := Value.WORD_T; END_IF
	VAR_TYPES.DWORD_T:
		CheckDeltaValue := ABS(DWORD_TO_LINT(LastValue.DWORD_T) - DWORD_TO_LINT(Value.DWORD_T)) >= DeltaVar;
		IF CheckDeltaValue THEN LastValue.DWORD_T := Value.DWORD_T; END_IF
	VAR_TYPES.LWORD_T:
	//here we use no expand but check min max because no bigger data type...
		IF LastValue.LWORD_T <= Value.LWORD_T THEN
			CheckDeltaValue := Value.LWORD_T - LastValue.LWORD_T >= UINT_TO_ULINT(DeltaVar);	
		ELSE
			CheckDeltaValue := LastValue.LWORD_T - Value.LWORD_T >= UINT_TO_ULINT(DeltaVar);
		END_IF
		IF CheckDeltaValue THEN LastValue.LWORD_T := Value.LWORD_T; END_IF
	VAR_TYPES.DATE_T:
		CheckDeltaValue := ABS(DATE_TO_LINT(LastValue.DATE_T) - DATE_TO_LINT(Value.DATE_T)) >= DeltaVar;
		IF CheckDeltaValue THEN LastValue.DATE_T := Value.DATE_T; END_IF
		
END_CASE

END_FUNCTION

// Common/Functions/GetValueFromPointer
FUNCTION GetValueFromPointer :  ALL_TYPES_UNION
VAR_INPUT
	PointerToValue:ALL_TYPES_UNION_POINTER;
	TypeOfValue: VAR_TYPES;
END_VAR
VAR
END_VAR

(*	SINT_T, USINT_T, INT_T, UINT_T, DINT_T, UDINT_T, 
				LINT_T, ULINT_T, REALT_T, LREAL_T*)
CASE TypeOfValue OF
	VAR_TYPES.SINT_T:
		GetValueFromPointer.SINT_T := PointerToValue.POINTER_TO_SINT_T^;
	VAR_TYPES.USINT_T:
		GetValueFromPointer.USINT_T := PointerToValue.POINTER_TO_USINT_T^;
	VAR_TYPES.INT_T:
		GetValueFromPointer.INT_T := PointerToValue.POINTER_TO_INT_T^;
	VAR_TYPES.UINT_T:
		GetValueFromPointer.UINT_T := PointerToValue.POINTER_TO_UINT_T^;
	VAR_TYPES.DINT_T:
		GetValueFromPointer.DINT_T := PointerToValue.POINTER_TO_DINT_T^;
	VAR_TYPES.UDINT_T:
		GetValueFromPointer.UDINT_T := PointerToValue.POINTER_TO_UDINT_T^;
	VAR_TYPES.LINT_T:
		GetValueFromPointer.LINT_T := PointerToValue.POINTER_TO_LINT_T^;
	VAR_TYPES.ULINT_T:
		GetValueFromPointer.ULINT_T := PointerToValue.POINTER_TO_ULINT_T^;
	VAR_TYPES.REAL_T:
		GetValueFromPointer.REAL_T := PointerToValue.POINTER_TO_REAL_T^;
	VAR_TYPES.LREAL_T:
		GetValueFromPointer.LREAL_T := PointerToValue.POINTER_TO_LREAL_T^;
	VAR_TYPES.BYTE_T:
		GetValueFromPointer.BYTE_T := PointerToValue.POINTER_TO_BYTE_T^;
	VAR_TYPES.WORD_T:
		GetValueFromPointer.WORD_T := PointerToValue.POINTER_TO_WORD_T^;
	VAR_TYPES.DWORD_T:
		GetValueFromPointer.DWORD_T := PointerToValue.POINTER_TO_DWORD_T^;
	VAR_TYPES.LWORD_T:
		GetValueFromPointer.LWORD_T := PointerToValue.POINTER_TO_LWORD_T^;
	VAR_TYPES.DT_T:
		GetValueFromPointer.DT_T := PointerToValue.POINTER_TO_DT_T^;
	VAR_TYPES.TIME_T:
		GetValueFromPointer.TIME_T := PointerToValue.POINTER_TO_TIME_T^;
	VAR_TYPES.LTIME_T:
		GetValueFromPointer.LTIME_T := PointerToValue.POINTER_TO_LTIME_T^;
	VAR_TYPES.TOD_T:
		GetValueFromPointer.TOD_T := PointerToValue.POINTER_TO_TOD_T^;
	VAR_TYPES.BOOL_T:
		GetValueFromPointer.BOOL_T := PointerToValue.POINTER_TO_BOOL_T^;
	VAR_TYPES.DATE_T:
		GetValueFromPointer.DATE_T := PointerToValue.POINTER_TO_DATE_T^;
	
END_CASE

END_FUNCTION

// Common/Functions/GetValueString
FUNCTION GetValueString : STRING
VAR_INPUT
	VALUE:ALL_TYPES_UNION;
	TypeOfValue:VAR_TYPES;
	DecimalPlace:INT;
END_VAR
VAR
END_VAR

(*	SINT_T, USINT_T, INT_T, UINT_T, DINT_T, UDINT_T, 
				LINT_T, ULINT_T, REALT_T, LREAL_T*)
CASE TypeOfValue OF
	VAR_TYPES.SINT_T:
		GetValueString := SINT_TO_STRING(VALUE.SINT_T);
	VAR_TYPES.USINT_T:
		GetValueString := USINT_TO_STRING(VALUE.USINT_T);		
	VAR_TYPES.INT_T:
		GetValueString := INT_TO_STRING(VALUE.INT_T);
	VAR_TYPES.UINT_T:
		GetValueString := UINT_TO_STRING(VALUE.UINT_T);
	VAR_TYPES.DINT_T:
		GetValueString := DINT_TO_STRING(VALUE.DINT_T);
	VAR_TYPES.UDINT_T:
		GetValueString := UDINT_TO_STRING(VALUE.UDINT_T);
	VAR_TYPES.LINT_T:
		GetValueString := LINT_TO_STRING(VALUE.LINT_T);
	VAR_TYPES.ULINT_T:
		GetValueString := ULINT_TO_STRING(VALUE.ULINT_T);
	VAR_TYPES.REAL_T:
		GetValueString := OSCAT_BASIC.REAL_TO_STRF(VALUE.REAL_T ,DecimalPlace,'.');
	VAR_TYPES.LREAL_T:
		GetValueString := OSCAT_BASIC.LREAL_TO_STRF(VALUE.LREAL_T ,DecimalPlace,'.');
	VAR_TYPES.BYTE_T:
		GetValueString := BYTE_TO_STRING(VALUE.BYTE_T);
	VAR_TYPES.WORD_T:
		GetValueString := WORD_TO_STRING(VALUE.WORD_T);
	VAR_TYPES.DWORD_T:
		GetValueString := DWORD_TO_STRING(VALUE.DWORD_T);
	VAR_TYPES.LWORD_T:
		GetValueString := LWORD_TO_STRING(VALUE.LWORD_T);
	VAR_TYPES.DT_T:
		GetValueString := DT_TO_STRING(VALUE.DT_T);
	VAR_TYPES.TIME_T:
		GetValueString := TIME_TO_STRING(VALUE.TIME_T);
	VAR_TYPES.LTIME_T:
		GetValueString := LTIME_TO_STRING(VALUE.LTIME_T);
	VAR_TYPES.TOD_T:
		GetValueString := TOD_TO_STRING(VALUE.TOD_T);
	VAR_TYPES.BOOL_T:
		GetValueString := BOOL_TO_STRING(VALUE.BOOL_T);
	VAR_TYPES.DATE_T:
		GetValueString := DATE_TO_STRING(VALUE.DATE_T);

	
	
END_CASE

END_FUNCTION

// Common/Function Blocks/CounterToActuall
FUNCTION_BLOCK CounterToActuall
VAR_INPUT

END_VAR
VAR_OUTPUT
	//actuell consumtion
	Actuell:LREAL;
	//consumption of counter
	Counters:ARRAY[0..MyConstants.COUNTER_COUNT-1]OF LREAL;
	//consumption at reset
	CountersValueAtReset:ARRAY[0..MyConstants.COUNTER_COUNT-1]OF LREAL;
	//actuell average Value
	CountersAverageValue:ARRAY[0..MyConstants.COUNTER_COUNT-1]OF LREAL;
	//counts of impuls
	Counts:ARRAY[0..MyConstants.COUNTER_COUNT-1]OF LREAL;
END_VAR
VAR
	CounterFaktor:LREAL;
	//time base for Counter val in s
	CounterTimeBase:LREAL;
	//impulse of Counter
	Pulse:POINTER TO BOOL;
	LastImp:CAA.TICK;
	RTrig:R_TRIG;
	CounterResetPointer:ARRAY[0..MyConstants.COUNTER_COUNT-1] OF POINTER TO BOOL;
	CounterIsParam:ARRAY[0..MyConstants.COUNTER_COUNT-1] OF BOOL;
	CounterEdge:ARRAY[0..MyConstants.COUNTER_COUNT-1]OF R_TRIG;
	i:UINT;
END_VAR

RTrig(CLK:= Pulse^);
IF RTrig.Q THEN
	Actuell := (CounterFaktor * CounterTimeBase) / (TO_LREAL(TICKS.GetTick(xDummy:= TRUE) - LastImp)/1000);
	LastImp := TICKS.GetTick(xDummy:= TRUE);
	//increase counters
	FOR i:=0 TO MyConstants.COUNTER_COUNT -1 DO
		Counters[i] := Counters[i] + CounterFaktor;
		Counts[i] := Counts[i] + 1;
		CountersAverageValue[i] := Counters[i] / Counts[i];  
	END_FOR
END_IF
//check if i have to reset counters....
FOR i:=0 TO MyConstants.COUNTER_COUNT -1 DO
	IF CounterIsParam[i] THEN
		CounterEdge[i](CLK:= CounterResetPointer[i]^);
		IF CounterEdge[i].Q THEN
			CountersValueAtReset[i] := Counters[i];
			Counters[i] := 0;
			Counts[i] := 0;
		END_IF
	END_IF
END_FOR

METHOD CounterInit
VAR_INPUT
	CounterFaktor:LREAL;
	//time base for Counter val in s
	CounterTimeBase:LREAL;
	//impulse of Counter
	Pulse:POINTER TO BOOL;
END_VAR
THIS^.CounterFaktor := CounterFaktor;
	
THIS^.CounterTimeBase := CounterTimeBase;

THIS^.Pulse :=	Pulse;
END_METHOD

METHOD SetCounterResetImp
VAR_INPUT
ImpVar:POINTER TO BOOL;
CounterNum:UINT;

END_VAR
IF  CounterNum < MyConstants.COUNTER_COUNT - 1 THEN
	CounterResetPointer[CounterNum] := ImpVar;
	CounterIsParam[CounterNum] := TRUE;
END_IF
END_METHOD

END_FUNCTION_BLOCK

// Common/Functions/test
FUNCTION test : bool
VAR_INPUT
END_VAR
VAR
	un:ALL_TYPES_UNION_POINTER:=(POINTER_TO_LREAL_T:=ADR(r1));
	
	r1:LREAL;
	//ar1:ARRAY[0..5] OF ALL_TYPES_UNION_POINTER[(ADR(r1))];
	
	pw1:PWConfigs:=(PointerTo:=( POINTER_TO_LREAL_T:=ADR(r1)));
	apw1:ARRAY[0..1]OF PWConfigs:=[(PointerTo:=( POINTER_TO_LREAL_T:=ADR(r1)))];
END_VAR

END_FUNCTION

// Common/Functions/StrEquals
//returns true if strings equals, else false
FUNCTION StrEquals : bool
VAR_INPUT
	str1:POINTER TO STRING;
	str2:POINTER TO STRING;
END_VAR
VAR
	
	pt1:POINTER TO BYTE;
	pt2:POINTER TO BYTE;
END_VAR

StrEquals := TRUE;

pt1 := str1;
pt2 := str2;
WHILE pt1^ <> 0 DO 
	IF pt1^ <> pt2^ THEN
		StrEquals := FALSE;
		EXIT;
	END_IF
	pt1 := pt1 + SIZEOF(BYTE);
	pt2 := pt2 + SIZEOF(BYTE);
END_WHILE
//check if string 2 ist at end to, if not, so not equal

IF pt2^ <> 0 THEN
	StrEquals := FALSE;
END_IF

END_FUNCTION

// Common/Functions/StrEqualsAtStart
//returns true if strings equals, else false
FUNCTION StrEqualsAtStart : bool
VAR_INPUT
	//needs to be the shorter string, this is the depending lenght
	str1:POINTER TO STRING;
	//scond String, is longer one with to check
	str2:POINTER TO STRING;
END_VAR
VAR
	
	pt1:POINTER TO BYTE;
	pt2:POINTER TO BYTE;
END_VAR

StrEqualsAtStart := TRUE;

pt1 := str1;
pt2 := str2;
WHILE pt1^ <> 0 DO 
	IF pt1^ <> pt2^ THEN
		StrEqualsAtStart := FALSE;
		EXIT;
	END_IF
	pt1 := pt1 + SIZEOF(BYTE);
	pt2 := pt2 + SIZEOF(BYTE);
END_WHILE

END_FUNCTION

// Common/Functions/GetValueFromStringPt
FUNCTION GetValueFromStringPt : BOOL
VAR_INPUT
	//type of var
	TypeOfValue:VAR_TYPES;
	//pointer to target
	Target:ALL_TYPES_UNION_POINTER;
	
	//value as string
	str:POINTER TO STRING(2000);
	
END_VAR
VAR
END_VAR

(*	SINT_T, USINT_T, INT_T, UINT_T, DINT_T, UDINT_T, 
				LINT_T, ULINT_T, REALT_T, LREAL_T*)
CASE TypeOfValue OF
	VAR_TYPES.SINT_T:
		Target.POINTER_TO_SINT_T^ := STRING_TO_SINT(str^);
	VAR_TYPES.USINT_T:
		Target.POINTER_TO_USINT_T^ := STRING_TO_USINT(str^);		
	VAR_TYPES.INT_T:
		Target.POINTER_TO_INT_T^ := STRING_TO_INT(str^);
	VAR_TYPES.UINT_T:
		Target.POINTER_TO_UINT_T^ := STRING_TO_UINT(str^);
	VAR_TYPES.DINT_T:
		Target.POINTER_TO_DINT_T^ := STRING_TO_DINT(str^);
	VAR_TYPES.UDINT_T:
		Target.POINTER_TO_UDINT_T^ := STRING_TO_UDINT(str^);
	VAR_TYPES.LINT_T:
		AtomicWriteLInt(pDest:= Target.POINTER_TO_LINT_T, liValue:= STRING_TO_LINT(str^));
		//Target.POINTER_TO_LINT_T^ := STRING_TO_LINT(str^);
	VAR_TYPES.ULINT_T:
		AtomicWriteULInt(pDest:= Target.POINTER_TO_ULINT_T, uliValue:= STRING_TO_ULINT(str^));
		//Target.POINTER_TO_ULINT_T^ := STRING_TO_ULINT(str^);
	VAR_TYPES.REAL_T:
		Target.POINTER_TO_REAL_T^ := STRING_TO_REAL(str^);
	VAR_TYPES.LREAL_T:
		AtomicWriteLReal(pDest:= Target.POINTER_TO_LREAL_T, lrValue:= STRING_TO_LREAL(str^));
		//Target.POINTER_TO_LREAL_T^ := STRING_TO_LREAL(str^);
	VAR_TYPES.BYTE_T:
		Target.POINTER_TO_BYTE_T^ := STRING_TO_BYTE(str^);
	VAR_TYPES.WORD_T:
		Target.POINTER_TO_WORD_T^ := STRING_TO_WORD(str^);
	VAR_TYPES.DWORD_T:
		Target.POINTER_TO_DWORD_T^ := STRING_TO_DWORD(str^);
	VAR_TYPES.LWORD_T:
		AtomicWriteLWord(pDest:= Target.POINTER_TO_LWORD_T, lwValue:= STRING_TO_LWORD(str^));
		//Target.POINTER_TO_LWORD_T^ := STRING_TO_LWORD(str^);
	VAR_TYPES.DT_T:
		Target.POINTER_TO_DT_T^ := STRING_TO_DT(str^);
	VAR_TYPES.TIME_T:
		Target.POINTER_TO_TIME_T^ := STRING_TO_TIME(str^);
	VAR_TYPES.LTIME_T:
		AtomicWriteLTime(pDest:= Target.POINTER_TO_LTIME_T, ltValue:= STRING_TO_LTIME(str^));
		//Target.POINTER_TO_TIME_T^ := STRING_TO_TIME(str^);
	VAR_TYPES.TOD_T:
		Target.POINTER_TO_TOD_T^ := STRING_TO_TOD(str^);
	VAR_TYPES.BOOL_T:
		Target.POINTER_TO_BOOL_T^ := STRING_TO_BOOL(str^);
	VAR_TYPES.DATE_T:
		Target.POINTER_TO_DATE_T^ := STRING_TO_DATE(str^);
	VAR_TYPES.STRING_T:
		Target.POINTER_TO_STRING_T^ := str^;
	
END_CASE

END_FUNCTION

// Common/Functions/StrEqualsAtStartWithDelimiter
//returns true if string at start equals and next char in string 2 is delim chart, else false
FUNCTION StrEqualsAtStartWithDelimiter : bool
VAR_INPUT
	//needs to be the shorter string, this is the depending lenght
	str1:POINTER TO STRING;
	//scond String, is longer one with to check
	str2:POINTER TO STRING;
	//split char/ Delmiter
	delimiter : BYTE;
END_VAR
VAR
	
	pt1:POINTER TO BYTE;
	pt2:POINTER TO BYTE;
END_VAR

StrEqualsAtStartWithDelimiter := TRUE;

pt1 := str1;
pt2 := str2;
WHILE pt1^ <> 0 AND pt2^<> 0 DO 
	IF pt1^ <> pt2^ THEN
		StrEqualsAtStartWithDelimiter := FALSE;
		EXIT;
	END_IF
	pt1 := pt1 + SIZEOF(BYTE);
	pt2 := pt2 + SIZEOF(BYTE);
END_WHILE
IF pt2^ <> delimiter THEN
	StrEqualsAtStartWithDelimiter := FALSE;
END_IF

END_FUNCTION

// Common/Functions/FindLastDot
FUNCTION FindLastDot : POINTER TO STRING(255)
VAR_INPUT
	str:POINTER TO STRING;
END_VAR
VAR
	pt:POINTER TO BYTE;
	c:BYTE;
END_VAR

c := GetChar('.');

pt := str;

WHILE pt^ <> 0 DO
	IF pt^ = c THEN
		FindLastDot := pt;
	END_IF
	pt := pt + SIZEOF(BYTE);
END_WHILE

END_FUNCTION

// Common/Functions/MakeAllTypesPointer
//returns a ALL_TYPES_UNION_POINTER from a dedicatet union

FUNCTION MakeAllTypesPointer : ALL_TYPES_UNION_POINTER
VAR_INPUT
	myType:VAR_TYPES;
	fromWho:POINTER TO ALL_TYPES_UNION;
END_VAR
VAR
END_VAR

CASE myType OF
	VAR_TYPES.SINT_T:
		MakeAllTypesPointer.POINTER_TO_SINT_T := ADR(fromWho^.SINT_T);
	VAR_TYPES.USINT_T:
		MakeAllTypesPointer.POINTER_TO_USINT_T := ADR(fromWho^.USINT_T);
	VAR_TYPES.INT_T:
		MakeAllTypesPointer.POINTER_TO_INT_T := ADR(fromWho^.INT_T);
	VAR_TYPES.UINT_T:
		MakeAllTypesPointer.POINTER_TO_UINT_T := ADR(fromWho^.UINT_T);
	VAR_TYPES.DINT_T:
		MakeAllTypesPointer.POINTER_TO_DINT_T := ADR(fromWho^.DINT_T);
	VAR_TYPES.UDINT_T:
		MakeAllTypesPointer.POINTER_TO_UDINT_T := ADR(fromWho^.UDINT_T);
	VAR_TYPES.LINT_T:
		MakeAllTypesPointer.POINTER_TO_LINT_T := ADR(fromWho^.LINT_T);
	VAR_TYPES.ULINT_T:
		MakeAllTypesPointer.POINTER_TO_ULINT_T := ADR(fromWho^.ULINT_T);
	VAR_TYPES.REAL_T:
		MakeAllTypesPointer.POINTER_TO_REAL_T := ADR(fromWho^.REAL_T);
	VAR_TYPES.LREAL_T:
		MakeAllTypesPointer.POINTER_TO_LREAL_T := ADR(fromWho^.LREAL_T);
	VAR_TYPES.BYTE_T:
		MakeAllTypesPointer.POINTER_TO_BYTE_T := ADR(fromWho^.BYTE_T);
	VAR_TYPES.WORD_T:
		MakeAllTypesPointer.POINTER_TO_WORD_T := ADR(fromWho^.WORD_T);
	VAR_TYPES.DWORD_T:
		MakeAllTypesPointer.POINTER_TO_DWORD_T := ADR(fromWho^.DWORD_T);
	VAR_TYPES.LWORD_T:
		MakeAllTypesPointer.POINTER_TO_LWORD_T := ADR(fromWho^.LWORD_T);
	VAR_TYPES.DT_T:
		MakeAllTypesPointer.POINTER_TO_DT_T := ADR(fromWho^.DT_T);
	VAR_TYPES.TIME_T:
		MakeAllTypesPointer.POINTER_TO_TIME_T := ADR(fromWho^.TIME_T);
	VAR_TYPES.TOD_T:
		MakeAllTypesPointer.POINTER_TO_TOD_T := ADR(fromWho^.TOD_T);
	VAR_TYPES.BOOL_T:
		MakeAllTypesPointer.POINTER_TO_BOOL_T := ADR(fromWho^.BOOL_T);
	VAR_TYPES.DATE_T:
		MakeAllTypesPointer.POINTER_TO_DATE_T := ADR(fromWho^.DATE_T);
	
END_CASE

END_FUNCTION

// Common/Function Blocks/StringImpact
FUNCTION_BLOCK StringImpact
VAR_INPUT
END_VAR
VAR_OUTPUT
END_VAR
VAR
	s1:STRING(10):='ABCDEFGHIJ';
	s2:STRING(5);
	s3:STRING(5);
	p1:POINTER TO STRING(10);
	p2:POINTER TO STRING(10);
END_VAR

p1 := ADR(s1);
p2 := ADR(s2);
p2^:= p1^;

END_FUNCTION_BLOCK

// Common/Function Blocks/GetInstanceName
{attribute 'reflection'}
FUNCTION_BLOCK GetInstanceName

//this is needed for FBinstance name in Variable
VAR_INPUT
END_VAR
VAR_OUTPUT
END_VAR
VAR
	{attribute 'instance-path'}
	{attribute 'noinit'}
	instanceName: STRING(255);//this string contains the instance name of the FB
	//here we get the "lowest" element of the name...
END_VAR

(*returns the instancename of calling instance as MQTT topic,
works only with string length < 255*)
METHOD GetInstanceTopic : string(255)
VAR_INPUT
END_VAR
VAR
	StrPt:POINTER TO BYTE;
END_VAR
GetInstanceTopic := instanceName;
//now delete last instance --> this

StrPt := FindLastDot(str:= ADR(GetInstanceTopic));
StrPt^ := 0; 

//now replace all  dots with "/"

GetInstanceTopic := OSCAT_BASIC.REPLACE_ALL(str:= GetInstanceTopic, src:= '.', rep:= '/');
//done...
END_METHOD

METHOD ReduceToLastNLevels : STRING(255)
VAR_INPUT
	Level:USINT;
END_VAR
VAR
	
	cmpByte:BYTE;
	bytePointer:POINTER TO BYTE;
	StringPointer:POINTER TO STRING;
	i:UINT;
END_VAR

cmpByte:= GetChar('.');

ReduceToLastNLevels := instanceName;

bytePointer :=  FindLastDot(str:= ADR(ReduceToLastNLevels));
bytePointer^ := 0;
//bytePointer := ADR(ReduceToLastNLevels) + len(str:= ADR(ReduceToLastNLevels));
bytePointer := bytePointer - 1;
i := 0;

WHILE bytePointer >= ADR(ReduceToLastNLevels) DO
	IF bytePointer^ = cmpByte THEN
		i := i + 1; 
	END_IF
	
	IF i = Level THEN
		
		StringPointer := bytePointer + 1;
		ReduceToLastNLevels := StringPointer^; 
		RETURN;
	END_IF
	bytePointer := bytePointer - 1;
END_WHILE
END_METHOD

END_FUNCTION_BLOCK

// Common/Functions/GetJSONValue
FUNCTION GetJSONValue : string(255)
VAR_INPUT
	fromWhere:POINTER TO STRING(65000);
END_VAR
VAR
	pt1: POINTER TO BYTE;
	pt2: POINTER TO BYTE;
	compByte1: BYTE;
	compByte2: BYTE;
	compByte3: BYTE;
END_VAR

// first find :

compByte1 := GetChar(':');
compByte2 := GetChar('"');
compByte3 := GetChar('}');

WHILE pt1^ <> compByte1 DO 
	pt1 := pt1 + 1;
END_WHILE


//check if '"' is next 

pt1 := pt1 + 1;

IF pt1^ = GetChar('"') THEN
	//add a 1
	pt1 := pt1 + 1;
END_IF

//here search for ',' or '}' or '"'

pt2 := pt1;

WHILE pt2^ <> compByte1 AND pt2^ <> compByte2 AND pt2^ <> compByte3 DO 
	pt2 := pt2 + 1;
END_WHILE

//so now we can copy the string...

SysMemCpy(pDest:= ADR(GetJSONValue), pSrc:= pt1, udiCount:= pt2 - pt1);
//now add trailing zero

pt2 := pt2 + 1;
pt2^:= 0;

END_FUNCTION

// Common/Function Blocks/RELAIS_OUT_16_TRANSLATOR
FUNCTION_BLOCK RELAIS_OUT_16_TRANSLATOR
VAR_INPUT
	outs:ARRAY[0..1] OF BYTE;
	target:POINTER TO ARRAY[0..1] OF BYTE;//I2C_MUX.PCF8575OUT;
END_VAR
VAR_OUTPUT
END_VAR
VAR
	temp0 : BYTE;
	temp1 : BYTE;
END_VAR
(*
translates data to an 16 bit relais output
output:
channel - bit
16 0.0
14 0.1
12 0.2
10 0.3
8 0.4
6 0.5
4 0.6
2 0.7
1 1.0
3 1.1
5 1.2
7 1.3
9 1.4
11 1.5
13 1.6
15 1.7

*)

temp0 := NOT outs[0];
temp1 := NOT outs[1];
target^[0].0 :=temp1.7;
target^[0].1 :=temp1.5;
target^[0].2 :=temp1.3;
target^[0].3 :=temp1.1;
target^[0].4 :=temp0.7;
target^[0].5 :=temp0.5;
target^[0].6 :=temp0.3;
target^[0].7 :=temp0.1;

target^[1].0 :=temp0.0;
target^[1].1 :=temp0.2;
target^[1].2 :=temp0.4;
target^[1].3 :=temp0.6;
target^[1].4 :=temp1.0;
target^[1].5 :=temp1.2;
target^[1].6 :=temp1.4;
target^[1].7 :=temp1.6;

END_FUNCTION_BLOCK

// Common/Function Blocks/SmartDim
FUNCTION_BLOCK SmartDim
VAR_INPUT
	start:BOOL;
	delayUntilDown:TIME;
	DataUp:POINTER TO SMART_DIMM;
	DataDown:POINTER TO SMART_DIMM;
END_VAR
VAR_OUTPUT
END_VAR
VAR
	aktStage:USINT;
	timerUntilOff:tof;
	LastTime:UINT;
	isOn: BOOL;
	StageTimer:ton;
	tmpOut:REAL;
END_VAR


IF start THEN
	IF NOT isOn THEN
		StageTimer(IN:= TRUE, PT:= DataUp^.values[aktStage].RunTime);
		tmpOut := OSCAT_BASIC.SCALE_R(
			X:= TO_REAL(StageTimer.ET), 
			I_LO:= DataUp^.values[aktStage]._from, 
			I_HI:= DataUp^.values[aktStage]._to, 
			O_LO:= DataUp^.values[aktStage]._from, 
			O_HI:= DataUp^.values[aktStage]._to);
	
	END_IF
	

END_IF

IF NOT isOn THEN
	;
END_IF

END_FUNCTION_BLOCK

// Common/Functions/Steps
FUNCTION Steps : real
VAR_INPUT
	aktVal:REAL;
	lastVal:REAL;
	stepsIn:REAL;
	base:REAL;
	mode: BOOL;//true --> up, false --> down
	
END_VAR
VAR
	aktFaktor:INT;
END_VAR

IF mode THEN
	aktFaktor := TO_INT((aktVal - base) / stepsIn);
	IF aktFaktor * StepsIn + base > aktVal THEN
		Steps := aktVal;
	ELSE
		Steps := lastVal;
	END_IF
ELSE
	;
END_IF

END_FUNCTION

// Common/Function Blocks/Spratzel
FUNCTION_BLOCK Spratzel
VAR_INPUT
	on: BOOL;
	onSpratzel:BOOL:=FALSE;
END_VAR
VAR_OUTPUT
	//otuput
	Out: BOOL;
	//spratzel is on
	isOn: BOOL;

END_VAR
VAR
	myRand:Rand;
	spratzelCount:INT;
	//aktuelle anzahl Spratzel
	aktSpratzel:INT;
	step:INT;
	start:r_trig;
	stop:f_trig;
	verz:ton;
	verzZeit:TIME;
	startTimer: BOOL;

END_VAR

start(clk:= on);
stop(clk:= on);
IF start.Q THEN
	step :=5;
	//anzahl der Spratzels ermitteln
	spratzelCount := myRand.getRand(HighIn:= 4, LowIn:= 1);
	verzZeit := INT_TO_TIME(myRand.getRand(HighIn:= 800, LowIn:= 100));
	startTimer := TRUE;
	aktSpratzel := 0;
END_IF
IF stop.Q THEN
	step := 0;
	out := FALSE;
	isOn := FALSE;
END_IF

verz(IN:= startTimer, pt:= verzZeit);
CASE step OF
	5:
	IF verz.Q THEN
		IF aktSpratzel >= spratzelCount THEN
			verz(IN:= FALSE, pt:= verzZeit);
			step := 15;
			isOn := TRUE;
			startTimer := FALSE;
		ELSE
			verz(IN:= FALSE, pt:= verzZeit);
			verzZeit := INT_TO_TIME(myRand.getRand(HighIn:= 800, LowIn:= 100));
			step := 10;
		END_IF
		out := TRUE;
	END_IF
	10:
	IF verz.Q THEN
		verz(IN:= FALSE, pt:= verzZeit);
		verzZeit := INT_TO_TIME(myRand.getRand(HighIn:= 800, LowIn:= 100));
		out := FALSE;
		step := 5;
		aktSpratzel := aktSpratzel + 1;
	END_IF
	15:
		;
END_CASE

METHOD setRand
VAR_INPUT
	newRand:Rand;
END_VAR
myRand := newRand;
END_METHOD

END_FUNCTION_BLOCK

// Common/Function Blocks/Rand
FUNCTION_BLOCK Rand
VAR_INPUT
END_VAR
VAR_OUTPUT
END_VAR
VAR
	myLast:INT;
END_VAR

METHOD getRand : INT
VAR_INPUT
	HighIn:INT;
	LowIn:int;
END_VAR
getRand := OSCAT_BASIC.RDM2(last:= MyLast, low:= HighIn, high:= LowIn);
END_METHOD

END_FUNCTION_BLOCK
